// TIA Portal project "SequencialMotorStarter" (V15)
// Sequencial Motor Starter. object oriented program mit SCL.

(* hardware
DEVICE "S71500/ET200MP station_1"  S7-1500 station
   slot 0: "Rail_0"  Rack  6ES7 590-1***0-0AA0
   slot 1: "PLC_1"  CPU 1512C-1 PN  6ES7 512-1CK01-0AB0  V2.5
      slot 3: "CPU display_1"  6ES7591-1AA00-0AA0
DEVICE "HMI_1"  TP900 Comfort
   slot 0: "HMI_1"  TP900 Comfort  6AV2 124-0JC01-0AX0  15.0.0.0
   slot 1: "HMI_RT_1"  TP900 Comfort  6AV2 124-0JC01-0AX0  15.0.0.0
   slot 5: "HMI_1.IE_CP_1"  PROFINET Interface  15.0.0.0
      slot 1: "PROFINET Interface_1"  PROFINET Interface
         slot 1: "Port_1"  Port
         slot 2: "Port_2"  Port
   slot 7: "HMI_1.MPI/DP_CP_1"  MPI/DP Interface  15.0.0.0
*)

// ===== PLC "PLC_1"  CPU 1512C-1 PN =====

TYPE "MotorI"
   STRUCT
      MotorI : Struct
         Start : Bool;
         Stop : Bool;
         Overload : Bool;
         WaitTime : Time := t#0s;
      END_STRUCT;
   END_STRUCT;
END_TYPE

TYPE "MotorO"
   STRUCT
      MotorO : Struct
         Coil : Bool;
      END_STRUCT;
   END_STRUCT;
END_TYPE

DATA_BLOCK "104_Program_DB"   // DB2
{ S7_Optimized_Access := 'FALSE' }
VERSION : 0.1
// stored: InstanceOfName 104_Program
"104_Program"
BEGIN
END_DATA_BLOCK

DATA_BLOCK "501_Data_block_1"   // DB501
{ S7_Optimized_Access := 'TRUE' }
VERSION : 0.1
   VAR
      MotorInput : Array[1..5] of "MotorI";
      MotorOutput : Array[1..5] of "MotorO";
      WaitTimer : TON_TIME;
   END_VAR
BEGIN
END_DATA_BLOCK

FUNCTION_BLOCK "101_SET_RESET"   // FB101, SCL
{ S7_Optimized_Access := 'TRUE' }
VERSION : 0.1
   VAR_INPUT
      set : Bool;
      reset : Bool;
   END_VAR
   VAR_OUTPUT
      Q1 : Bool;
   END_VAR
   VAR
      r_trig_set : R_TRIG;
      r_trig_reset : R_TRIG;
   END_VAR
BEGIN
   IF #reset = TRUE THEN
       #Q1 := FALSE;
   ELSIF #set = TRUE THEN
       #Q1 := TRUE;
   END_IF;
END_FUNCTION_BLOCK

FUNCTION_BLOCK "102_MotorEquip"   // FB102, SCL
{ S7_Optimized_Access := 'FALSE' }
VERSION : 0.1
   VAR_INPUT
      MotorInput : "MotorI";
   END_VAR
   VAR_OUTPUT
      MotorOutput : "MotorO";
   END_VAR
   VAR
      WaitTimer : TON_TIME;
      RS_Output : Bool;
   END_VAR
   // WaitTimer.PT := T#0MS;
BEGIN
   (*
   "10_SET_RESET_DB"(set := #MotorInput.MotorI.Start,
                     reset := #MotorInput.MotorI.Stop,
                     Q1 => #RS_Output);
   *)
   "201_Set_Reset"(set:=#MotorInput.MotorI.Start,
                  reset:=#MotorInput.MotorI.Stop,
                  Q1=>#RS_Output);

   IF #RS_Output = TRUE AND #MotorInput.MotorI.Overload = FALSE THEN  /////////Check if start input is activated , and there is no overload or stop button activated
       #WaitTimer(IN := TRUE,
                  PT := #MotorInput.MotorI.WaitTime);  ////Init the timer according to the presetTime provided and activate the timer
       //
       IF #WaitTimer.Q THEN                     /////////If preset Time elapses turn on the motor
           #MotorOutput.MotorO.Coil := TRUE;
           #WaitTimer(IN := False,
                      PT := t#0s);
       END_IF;
   END_IF;

   IF #MotorInput.MotorI.Stop OR #MotorInput.MotorI.Overload THEN  ///////////If there is a stop or an overload , or start input is deactivaed , turn off the motor and deactiavte the ditmer 
       #WaitTimer(IN := FALSE,
                  PT := t#0s);
       #MotorOutput.MotorO.Coil := FALSE;
   END_IF;
END_FUNCTION_BLOCK

FUNCTION_BLOCK "103_test_Program"   // FB103, SCL
{ S7_Optimized_Access := 'TRUE' }
VERSION : 0.1
   VAR
      MotorInput : Array[1..#NUM_MOTORS] of "MotorI";
      MotorOutput : Array[1..#NUM_MOTORS] of "MotorO";
      Motors : Array[1..#NUM_MOTORS] of "102_MotorEquip";
      SerialIndex : Int := 1;
      Index : Int;
      GeneralStart : Bool;
      GeneralStop : Bool;
      ResetFault : Bool;
      FaultMotorNumber : Int;
      Succed : Bool;
      Failed : Bool;
      StopTrig : R_TRIG;
      ResetTrig : R_TRIG;
   END_VAR
   VAR CONSTANT
      NUM_MOTORS : Int := 5;
   END_VAR
BEGIN
   /////////////////////////Assignment and Initialization/////////////////////////
   (*
   FOR #Index := 1 TO #NUM_MOTORS BY 1 DO
       #MotorInput[#Index].MotorI.Start := #GeneralStop;      ////Bind the stop button of all motors to one single General Stop                                               

       // this following binding doesn't work in Siemens, also calling a FB created 
       // from one instance of an array doesn't work.
       #Motors[#Index](MotorInput := #MotorInput[#Index],
                       MotorOutput => #MotorOutput[#Index]);
       //#MotorInput[#Index].MotorI.WaitTime := T#5S;           ///////////Assign Wait time for all motors to be 3seconds                                
   END_FOR;
   *)

   (* try ------------------------
   FOR #Index := 1 TO #NUM_MOTORS-1 BY 1 DO
       #Motors[#Index].MotorInput.MotorI.Start := TRUE;
       IF #Motors[#Index].MotorOutput.MotorO.Coil = TRUE THEN
           #Succed := TRUE;
       END_IF;
   END_FOR;

   #MotorInput[1].MotorI.Start := TRUE;
   #MotorInput[2].MotorI.Start := TRUE;
   #MotorInput[3].MotorI.Start := TRUE;
   #MotorInput[4].MotorI.Start := TRUE;

   #Motors[1].MotorInput.MotorI.Start := #MotorInput[1].MotorI.Start;
   #MotorOutput[1].MotorO.Coil := #Motors[1].MotorOutput.MotorO.Coil;

   #MotorInput[1].MotorI.Start := #GeneralStart;
   IF #MotorOutput[1].MotorO.Coil THEN
       #MotorInput[2].MotorI.Start := TRUE;
   END_IF;
   * try ------------------------*)

   (*
   /////////////////////////////Sequence OPeration///////////////
   #MotorInput[1].MotorI.Start := #GeneralStart; /////////////The first motor of the sequence should be assigned to the start button

   IF #MotorOutput[#SerialIndex].MotorO.Coil AND #Succed = FALSE AND #Failed = FALSE THEN   //////////////////Pressing the start button would yield the first motor in the sequence to be on 
       ////////////////////////////////////////////////////////////////////////////////////////// IF so , actuate the rest Of the  sequence
       IF #SerialIndex > #NUM_MOTORS THEN           //////Guard to prevent the SerialIndex from being assigned to values outside the bounds of the array
           #SerialIndex := 1;
       ELSE
           #SerialIndex := #SerialIndex + 1;                /////If the current motor coil is activated , activate the next motor in sequence
           #MotorInput[#SerialIndex].MotorI.Start := TRUE;
       END_IF;
   END_IF;

   IF #SerialIndex - 1 = #NUM_MOTORS THEN                   ////When we have looped thorugh all motors , set a "Succed" flag and reset the SerialIndex to 1 .
       #Succed := TRUE;
       #SerialIndex := 1;
   END_IF;

   ///////////////////////////////////Handling a General Stop////////////////
   #StopTrig(CLK := #GeneralStop);
   IF #StopTrig.Q THEN        /////If a general Stop is detected
       #Succed := FALSE;            /////Succed flag is set to FALSE
       FOR #Index := 1 TO #NUM_MOTORS BY 1 DO        ///// Deactivate all the Start Inputs for all motors
           #MotorInput[#Index].MotorI.Start := FALSE;
       END_FOR;
   END_IF;

   //////////////////////Handling Overloads/////////////////////////
   FOR #Index := 1 TO #NUM_MOTORS BY 1 DO     /////////////if there is ANY Overload fault then set the failed flag to TRUE
       IF #MotorInput[#Index].MotorI.Overload THEN
           #Failed := TRUE;
           #FaultMotorNumber := #Index;
           EXIT;
       END_IF;
   END_FOR;
   //////////////////////////////

   IF #Failed THEN ////////////////////// IF The failed flag is set to TRUE , assign FALSE To all start signals and assign a general stop
       FOR #Index := 1 TO #NUM_MOTORS BY 1 DO
           #MotorInput[#Index].MotorI.Start := FALSE;
           #GeneralStop := TRUE;
       END_FOR;
   END_IF;

   ///////////////////////////////////Reseting the fault
   #ResetTrig(CLK := #ResetFault);////////////////If a reset fault is detected , reset the FAILED flag and Set GeneralStop to False
   IF #ResetTrig.Q THEN
       #Failed := FALSE;
       #GeneralStop := FALSE;
       #SerialIndex := 1;
   END_IF;
   *)
END_FUNCTION_BLOCK

FUNCTION_BLOCK "104_Program"   // FB104, SCL
{ S7_Optimized_Access := 'FALSE' }
VERSION : 0.1
   VAR
      SerialIndex : Int := 1;
      Index : Int;
      GeneralStart : Bool;
      GeneralStop : Bool;
      ResetFault : Bool;
      FaultMotorNumber : Int;
      StartTrig_IN : Bool;
      StopTrig_In : Bool;
      ResetTrig_In : Bool;
      Succed : Bool;
      Failed : Bool;
      StartTrig : R_TRIG;
      StopTrig : R_TRIG;
      ResetTrig : R_TRIG;
      IWaitTime : Time := T#3s;
   END_VAR
   VAR CONSTANT
      NUM_MOTORS : Int := 5;
   END_VAR
BEGIN
   // alle werte von "WaitTime <-- MotorO" in alle Motoren Binden zu variable "IWaitTime" in diese FB  
   FOR #Index := 1 TO #NUM_MOTORS DO
       "501_Data_block_1".MotorInput[#Index].MotorI.WaitTime := #IWaitTime;
   END_FOR;

   // Ersten Maschine Starten button ist dem Starten punkt für alles nächsten Maschinen. 
   IF #GeneralStart = FALSE THEN
       #StartTrig(CLK := #StartTrig_IN OR "501_Data_block_1".MotorInput[1].MotorI.Start,
                  Q => #GeneralStart);
   END_IF;

   IF #GeneralStart=TRUE AND "501_Data_block_1".MotorOutput[1].MotorO.Coil=FALSE THEN
       "501_Data_block_1".MotorInput[1].MotorI.Start := TRUE;
       "202_MotorEquip"(MotorInput:="501_Data_block_1".MotorInput[1],
                    MotorOutput=>"501_Data_block_1".MotorOutput[1]);
   END_IF;

   // Wenn die erste Maschine erfolgreich startet, dann starten Sie die nächsten Maschinen nacheinander. 
   IF #GeneralStart=TRUE AND #SerialIndex<#NUM_MOTORS AND "501_Data_block_1".MotorOutput[#SerialIndex].MotorO.Coil = TRUE  THEN
       "501_Data_block_1".MotorInput[#SerialIndex+1].MotorI.Start := TRUE;
       "202_MotorEquip"(MotorInput := "501_Data_block_1".MotorInput[#SerialIndex+1],
                        MotorOutput => "501_Data_block_1".MotorOutput[#SerialIndex+1]);
       IF "501_Data_block_1".MotorOutput[#SerialIndex+1].MotorO.Coil = true THEN
           #SerialIndex:=#SerialIndex+1;
       END_IF;
   END_IF;

   // Überlastung des Motors bewältigen
   FOR #Index := 1 TO #NUM_MOTORS DO
       IF "501_Data_block_1".MotorInput[#Index].MotorI.Overload = TRUE THEN
           #GeneralStop:=TRUE;
           #FaultMotorNumber := #Index;
       END_IF;
   END_FOR;


   // Wann alles Machinen starten erfolgreich dann machen [Succed] flag True.
   IF "501_Data_block_1".MotorOutput[#NUM_MOTORS].MotorO.Coil = TRUE THEN
       #Failed := FALSE;
       #GeneralStart := FALSE;
       #Succed := TRUE;
       #SerialIndex := 1;
   END_IF;

   IF #GeneralStop = FALSE THEN
       #StopTrig(CLK := #StopTrig_In,
                  Q => #GeneralStop);
   END_IF;

   // Stoppen einer Maschine oder oveload signal von einer Maschine stoppt alle Maschinen.
   IF #GeneralStop = TRUE THEN
       FOR #Index := 1 TO #NUM_MOTORS DO
           "501_Data_block_1".MotorInput[#Index].MotorI.Start := FALSE;
           "501_Data_block_1".MotorInput[#Index].MotorI.Stop := TRUE;
           "202_MotorEquip"(MotorInput := "501_Data_block_1".MotorInput[#Index],
                            MotorOutput => "501_Data_block_1".MotorOutput[#Index]);
           #GeneralStart := FALSE;
           #Failed := TRUE;
           #Succed := FALSE;
       END_FOR;
   END_IF;
   #Index := 0;

   IF #ResetFault = FALSE THEN
       #ResetTrig(CLK := #ResetTrig_In,
                  Q => #ResetFault);
   END_IF;

   // RESET betrieb
   IF #ResetFault = TRUE THEN
       FOR #Index := 1 TO #NUM_MOTORS DO
           "501_Data_block_1".MotorInput[#Index].MotorI.Start := FALSE;
           "501_Data_block_1".MotorInput[#Index].MotorI.Stop := FALSE;
           "202_MotorEquip"(MotorInput := "501_Data_block_1".MotorInput[#Index],
                            MotorOutput => "501_Data_block_1".MotorOutput[#Index]);
           #GeneralStart := FALSE;
           #Failed := FALSE;
           #Succed := FALSE;
           #GeneralStop := FALSE;
           #FaultMotorNumber := 0;
       END_FOR;
   END_IF;
   #Index := 0;
   #ResetFault := False;
END_FUNCTION_BLOCK

FUNCTION "201_Set_Reset" : Void   // FC201, SCL
{ S7_Optimized_Access := 'TRUE' }
VERSION : 0.1
   VAR_INPUT
      set : Bool;
      reset : Bool;
   END_VAR
   VAR_OUTPUT
      Q1 : Bool;
   END_VAR
BEGIN
   IF #reset = TRUE THEN
       #Q1 := FALSE;
   ELSIF #set = TRUE THEN
       #Q1 := TRUE;
   END_IF;
END_FUNCTION

FUNCTION "202_MotorEquip" : Void   // FC202, SCL
{ S7_Optimized_Access := 'TRUE' }
VERSION : 0.1
   VAR_INPUT
      MotorInput : "MotorI";
   END_VAR
   VAR_OUTPUT
      MotorOutput : "MotorO";
   END_VAR
   VAR_TEMP
      RS_Output : Bool;
   END_VAR
BEGIN
   (*
   "10_SET_RESET_DB"(set := #MotorInput.MotorI.Start,
                     reset := #MotorInput.MotorI.Stop,
                     Q1 => #RS_Output);
   *)
   "201_Set_Reset"(set := #MotorInput.MotorI.Start,
                  reset := #MotorInput.MotorI.Stop,
                  Q1 => #RS_Output);

   IF #RS_Output = TRUE AND #MotorInput.MotorI.Overload = FALSE THEN  /////////Check if start input is activated , and there is no overload or stop button activated
       "501_Data_block_1".#WaitTimer(IN := TRUE,
                  PT := #MotorInput.MotorI.WaitTime);  ////Init the timer according to the presetTime provided and activate the timer
       //
       IF "501_Data_block_1".#WaitTimer.Q THEN                     /////////If preset Time elapses turn on the motor
           #MotorOutput.MotorO.Coil := TRUE;
           "501_Data_block_1".#WaitTimer(IN := False,
                      PT := t#0s);
       END_IF;
   END_IF;

   IF #MotorInput.MotorI.Stop OR #MotorInput.MotorI.Overload THEN  ///////////If there is a stop or an overload , or start input is deactivaed , turn off the motor and deactiavte the ditmer 
       "501_Data_block_1".#WaitTimer(IN := FALSE,
                  PT := t#0s);
       #MotorOutput.MotorO.Coil := FALSE;
   END_IF;
END_FUNCTION

ORGANIZATION_BLOCK "Main"   // OB1, LAD, ProgramCycle
TITLE = "Main Program Sweep (Cycle)"
{ S7_Optimized_Access := 'TRUE' }
VERSION : 0.1
   VAR_INPUT
      Initial_Call : Bool;   // Initial call of this OB
      Remanence : Bool;   // =True, if remanent data are available
   END_VAR
BEGIN

REGION Network 1
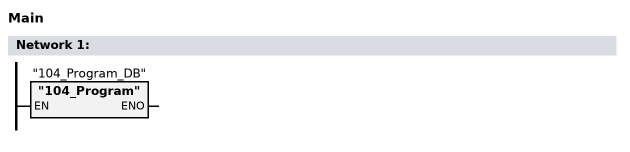
   RUNG wire#powerrail
      "104_Program_DB"()
   END_RUNG
   // the same network as SCL:
   "104_Program_DB"();   // "104_Program"
END_REGION
END_ORGANIZATION_BLOCK

(* ===== HMI "HMI_RT_1" =====
system functions are stored by id; their names below are inferred from use
connection "HMI_Connection_1": ETHERNET, S7_1500_OMS

HMI tags "Default tag table"
   "501_Data_block_1_MotorOutput{1}_MotorO_Coil" : Bool = PLC "501_Data_block_1".MotorOutput[1].MotorO.Coil, 1 s
   "501_Data_block_1_MotorOutput{2}_MotorO_Coil" : Bool = PLC "501_Data_block_1".MotorOutput[2].MotorO.Coil, 1 s
   "501_Data_block_1_MotorOutput{3}_MotorO_Coil" : Bool = PLC "501_Data_block_1".MotorOutput[3].MotorO.Coil, 1 s
   "501_Data_block_1_MotorOutput{4}_MotorO_Coil" : Bool = PLC "501_Data_block_1".MotorOutput[4].MotorO.Coil, 1 s
   "501_Data_block_1_MotorOutput{5}_MotorO_Coil" : Bool = PLC "501_Data_block_1".MotorOutput[5].MotorO.Coil, 1 s
   "104_Program_DB_StartTrig_IN" : Bool = PLC "104_Program_DB".StartTrig_IN AT %DB2.DBX8.0, 1 s
   "104_Program_DB_StopTrig_In" : Bool = PLC "104_Program_DB".StopTrig_In AT %DB2.DBX8.1, 1 s
   "104_Program_DB_ResetTrig_In" : Bool = PLC "104_Program_DB".ResetTrig_In AT %DB2.DBX8.2, 1 s
   "104_Program_DB_FaultMotorNumber" : Int = PLC "104_Program_DB".FaultMotorNumber AT %DB2.DBW6, 1 s
   "104_Program_DB_Succed" : Bool = PLC "104_Program_DB".Succed AT %DB2.DBX8.3, 1 s
   "104_Program_DB_Failed" : Bool = PLC "104_Program_DB".Failed AT %DB2.DBX8.4, 1 s

screen "Root screen" 800x444, template "Template_1"
   Button "Button_1" at 35,29 size 80x19; TextOff 'General Start'
      on Press: SetBit("104_Program_DB_StartTrig_IN")
      on Release: ResetBit("104_Program_DB_StartTrig_IN")
   Button "Button_2" at 35,53 size 80x19; TextOff 'General Stop'
      on Press: SetBit("104_Program_DB_StopTrig_In")
      on Release: ResetBit("104_Program_DB_StopTrig_In")
   Button "Button_3" at 35,77 size 80x19; TextOff 'Reset Fault'
      on Release: ResetBit("104_Program_DB_ResetTrig_In")
      on Press: SetBit("104_Program_DB_ResetTrig_In")
   Circle "Circle_1" at 136,24 size 24x24
      Appearance <- "104_Program_DB_Succed"
   Circle "Circle_2" at 136,56 size 24x24
      Appearance <- "104_Program_DB_Failed"
   TextField "Text field_1" at 168,24 size 53x20; Text 'Succeed'
   TextField "Text field_2" at 168,56 size 39x20; Text 'Failed'
   IOField "I/O field_1" at 133,87 size 32x32; FormatPattern 99
      ProcessValue <- "104_Program_DB_FaultMotorNumber"
   TextField "Text field_3" at 168,88 size 126x20; Text 'Overloaded motor no'
   GraphicView "Graphic view_1" at 316,16 size 408x376; Picture "imageedit_1_6157493393"
   Circle "Circle_3" at 689,79 size 24x24
      Visibility <- "501_Data_block_1_MotorOutput{2}_MotorO_Coil"
   Circle "Circle_4" at 655,184 size 24x24
      Visibility <- "501_Data_block_1_MotorOutput{4}_MotorO_Coil"
   Circle "Circle_5" at 416,184 size 24x24
      Visibility <- "501_Data_block_1_MotorOutput{3}_MotorO_Coil"
   Circle "Circle_6" at 448,80 size 24x24
      Visibility <- "501_Data_block_1_MotorOutput{1}_MotorO_Coil"
   Circle "Circle_7" at 528,360 size 24x24
      Visibility <- "501_Data_block_1_MotorOutput{5}_MotorO_Coil"

Template "Template_1" 800x444
   Button "Exit" at 750,407 size 49x35; TextOff 'Exit'; PictureOff "ExitRuntime_TP1500_Comfort_V2_TR"; PictureOn "ExitRuntime_TP1500_Comfort_V2_TR"
      on Release: StopRuntime(0)
   Button "Template_Button" at 700,407 size 49x35; TextOff 'Text'
   Button "Template_Button_1" at 650,407 size 49x35; TextOff 'Text'
   Button "Template_Button_2" at 600,407 size 49x35; TextOff 'Text'
   Button "Template_Button_3" at 550,407 size 49x35; TextOff 'Text'
   Button "Template_Button_4" at 500,407 size 49x35; TextOff 'Text'
   Button "Template_Button_5" at 450,407 size 49x35; TextOff 'Text'
   Button "Template_Button_6" at 400,407 size 49x35; TextOff 'Text'
   Button "Template_Button_7" at 351,407 size 49x35; TextOff 'Text'
   Button "Template_Button_8" at 301,407 size 49x35; TextOff 'Text'
   Button "Template_Button_9" at 251,407 size 49x35; TextOff 'Text'
   Button "Template_Button_10" at 201,407 size 49x35; TextOff 'Text'
   Button "Template_Button_11" at 151,407 size 49x35; TextOff 'Text'
   Button "Template_Button_12" at 101,407 size 49x35; TextOff 'Text'
   Button "Template_Button_13" at 51,407 size 49x35; TextOff 'Text'
   Button "Start screen" at 1,407 size 49x35; TextOff 'Start screen'; PictureOff "NavigateHome_TP1500_Comfort_V2_TR"; PictureOn "NavigateHome_TP1500_Comfort_V2_TR"
      on Release: ActivateScreen("Root screen", 0)
*)